(* CoDeSys 2.3 export: FBK16PUMPSTRAINING.EXP *)

(* POU K16/fbK16PumpsTraining, ST *)
FUNCTION_BLOCK fbK16PumpsTraining
(*
	Функция тренировки насосов К15
*)
VAR CONSTANT
	TrainingDelay: TIME := T#24h;		(*Задержка на включение тренировки*)
	TrainingPeriod: TIME := T#10s;	(*Период тренировки*)
END_VAR
VAR
	PumpOffDelay : ARRAY [1..MAX_K16_PUMPS_NUM] OF TON;
	PumpTrainingTimer : ARRAY [1..MAX_K16_PUMPS_NUM] OF TP;
END_VAR
VAR_TEMP
	i: USINT;
END_VAR
FOR i := 1 TO MAX_K16_PUMPS_NUM DO
	PumpOffDelay[i](IN := fGetK16Pump(i), PT := TrainingDelay);
	PumpTrainingTimer[i](IN := PumpOffDelay[i].Q, PT := TrainingPeriod);
	IF PumpTrainingTimer[i].Q THEN
		fTurnOnK16Pump(i);
	END_IF;
END_FOR;
END_FUNCTION_BLOCK
